FUNCTION Matrix_SubMatrix : Bool
VAR_INPUT
	M_Super : REFERENCE TO Matrix;
	M_Sub : REFERENCE TO Matrix;
	RowStart : UINT;
	RowCount : UINT;
	ColStart : UINT;
	ColCount : UINT;
END_VAR

VAR
	Ri : UINT;
	Ci : UINT;
END_VAR

IF RowStart + RowCount > M_Super.Rows OR ColStart + ColCount > M_Super.Cols THEN
	Matrix_SubMatrix := FALSE;
	RETURN;
END_IF
IF M_Sub.Rows <> RowCount  OR M_Sub.Cols <> ColCount THEN
	Matrix_SubMatrix := FALSE;
	RETURN;
END_IF

Matrix_SubMatrix := TRUE;

IF RowCount = 0 OR ColCount = 0 THEN
	RETURN;//valid to get a zero-len matrix as the result, but indexing below will cause a pagefault due to creating 32k+ warning messages for invalid access
END_IF

FOR Ri := 0 TO RowCount-1 DO
	FOR Ci := 0 TO ColCount-1 DO
		M_Sub.SetRC(Ri,Ci,M_Super.GetRC(RowStart+Ri,ColStart+Ci));
	END_FOR
END_FOR

END_FUNCTION

(* stored: Version 1.1.0.1, ProductVersion 3.1.4024.9
   POU Matrix_SubMatrix: Id {e584d28a-8010-4956-af80-0bbe9d155507}, SpecialFunc None *)
